// TIA Portal V17 export
// export: Created 2026-07-06T15:33:01.4639971Z, ExportSetting WithDefaults, DisplayName Totally Integrated Automation Portal, DisplayVersion V17, DisplayName TIA Portal Openness, DisplayVersion V17, DisplayName TIA Portal Version Control Interface, DisplayVersion V17, DisplayName STEP 7 Professional, DisplayVersion V17, DisplayName STEP 7 Safety, DisplayVersion V17, DisplayName WinCC Professional, DisplayVersion V17
FUNCTION_BLOCK "PULSE_TIMER"   // FB5, LAD
{ S7_Optimized_Access := 'TRUE' }
VERSION : 0.1
// stored: AutoNumber true, IsIECCheckEnabled false, IsRetainMemResEnabled false, MemoryReserve 100, SetENOAutomatically false, UDAEnableTagReadback false
   VAR_INPUT
      "PULSE HZ" : Real;
   END_VAR
   VAR_OUTPUT
      PULSE : Bool;
   END_VAR
   VAR
      Clock_Timer_1 : IEC_TIMER;
      Clock_Timer_2 : IEC_TIMER;
      "Time(s)" { S7_SetPoint := 'True'} : Real;
      "Time(ms)" : Real;
      "Time" : Int;
   END_VAR
BEGIN

REGION Network 1: Timer Loop
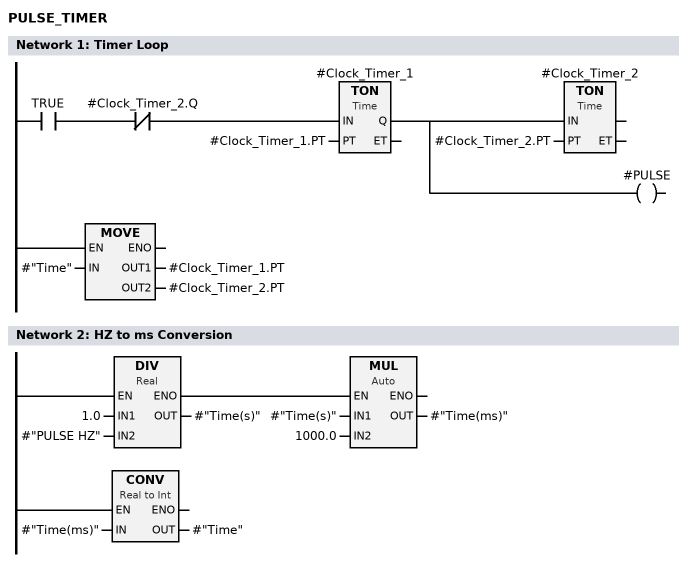
   RUNG wire#powerrail
      Contact( TRUE )
      I_Contact( #Clock_Timer_2.Q )
      { S7_Templates := "time_type := Time" } #Clock_Timer_1.TON(pt := #Clock_Timer_1.PT, et =>)
      wire#w1
      { S7_Templates := "time_type := Time" } #Clock_Timer_2.TON(pt := #Clock_Timer_2.PT, et =>)
   END_RUNG
   RUNG wire#w1
      Coil( #PULSE )
   END_RUNG
   RUNG wire#powerrail
      Move(in := #"Time", out1 => #Clock_Timer_1.PT, out2 => #Clock_Timer_2.PT)
   END_RUNG
   // the same network as SCL:
   #Clock_Timer_1.TON(IN := TRUE AND NOT #Clock_Timer_2.Q, PT := #Clock_Timer_1.PT);
   #Clock_Timer_2.TON(IN := #Clock_Timer_1.Q, PT := #Clock_Timer_2.PT);
   #PULSE := #Clock_Timer_1.Q;
   #Clock_Timer_1.PT := #"Time";
   #Clock_Timer_2.PT := #"Time";
END_REGION

REGION Network 2: HZ to ms Conversion
   RUNG wire#powerrail
      { S7_Templates := "SrcType := Real" } Div(in1 := 1.0, in2 := #"PULSE HZ", out => #"Time(s)")
      Mul(in1 := #"Time(s)", in2 := 1000.0, out => #"Time(ms)")
   END_RUNG
   RUNG wire#powerrail
      { S7_Templates := "[SrcType := Real, DestType := Int]" } Convert(in := #"Time(ms)", out => #"Time")
   END_RUNG
   // the same network as SCL:
   #"Time(s)" := 1.0 / #"PULSE HZ";
   #"Time(ms)" := #"Time(s)" * 1000.0;
   #"Time" := REAL_TO_INT(#"Time(ms)");
END_REGION
END_FUNCTION_BLOCK
